// TIA Portal V21 export
DATA_BLOCK "LCC_ConfigDevice_DB"   // DB2
AUTHOR : SIOS
FAMILY : LCC
VERSION : 1.0
// stored: InstanceOfName LCC_ConfigDevice, InstanceOfType FB
"LCC_ConfigDevice"
   // VAR_INPUT
   //    hwID : HW_IO;
   // END_VAR
   // VAR_OUTPUT
   //    statusID : USInt;
   //    status { ExternalAccessible := 'False'; ExternalVisible := 'False'; ExternalWritable := 'False'} : DWord;
   // END_VAR
   // VAR_IN_OUT
   //    dataRec : Variant;
   // END_VAR
   // VAR
   //    statReq : Bool;
   //    instWriteRecord { ExternalAccessible := 'False'; ExternalVisible := 'False'; ExternalWritable := 'False'; S7_SetPoint := 'True'} : WRREC;
   // END_VAR
BEGIN
END_DATA_BLOCK
